TYPE ST_TimeDiff :
STRUCT
	sSecond : WORD;
	mMillisecond : WORD;
END_STRUCT
END_TYPE

(* stored: Version 1.1.0.1, ProductVersion 3.1.4024.3
   DUT ST_TimeDiff: Id {ab07a440-c96d-4810-8ba0-5d8ad617de47} *)
